FUNCTION Lifting : INT
VAR_INPUT
	EndPosition: INT;
	State: INT;
END_VAR
VAR
	MovementEnum: Movement;
	NextState: INT;
	MotorDirectionEnum: MovementDirection;
END_VAR

IF Automatic.LiftingPositionAuto > EndPosition THEN
	MotorDirectionEnum := MovementDirection.TowardsSensor;
ELSE
	MotorDirectionEnum := MovementDirection.AwayFromSensor;
END_IF

IF MotorDirectionEnum = MovementDirection.TowardsSensor THEN
	IF Automatic.LiftingPositionAuto > EndPosition THEN
		IO.MotorLiftingDirection := (MotorDirectionEnum = MovementDirection.TowardsSensor);
		IF NOT Automatic.SafetyLON THEN
			Automatic.GCurrentlyMoving := TRUE;
			IO.MotorLifting := (MovementEnum = Movement.ON);
		END_IF
		NextState := State;
	ELSE
		IO.MotorLifting := (MovementEnum = Movement.OFF);
		NextState := State + 1;
		Automatic.LCurrentlyMoving := FALSE;
	END_IF
ELSE
	IF Automatic.LiftingPositionAuto < EndPosition THEN
		IO.MotorLiftingDirection := (MotorDirectionEnum = MovementDirection.AwayFromSensor);
		IF (NOT Automatic.SafetyLON) THEN
			Automatic.LCurrentlyMoving := TRUE;
			IO.MotorLifting := (MovementEnum = Movement.ON);
		END_IF
		NextState := State;
	ELSE
		IO.MotorLifting := (MovementEnum = Movement.OFF);
		NextState := State + 1;
		Automatic.LCurrentlyMoving := FALSE;
	END_IF
END_IF

Lifting := NextState;
RETURN;

END_FUNCTION

(* stored: Version 1.1.0.1, ProductVersion 3.1.4024.13
   POU Lifting: Id {8bb0c76d-ac8e-48ce-b59f-fd84e7697f93}, SpecialFunc None *)
